// TIA Portal V18 export
VAR_GLOBAL   // PLC tag table "Assigned IO"
   HPU_In AT %I0.0 : "Starter_HPU_IO_In";
   HPU_Out AT %Q0.0 : "Starter_HPU_IO_Out";
   Console_In AT %I200.0 : "Console_IO_In";
   Console_Out AT %Q200.0 : "Console_IO_Out";
   ComFault AT %M20.1 : Bool;
   SystemFault AT %M1.0 : Bool;
   RemConsole_In AT %I500.0 : "RemConsole_IO_In";
   RemConsole_Out AT %Q500.0 : "RemConsole_IO_Out";
   RemConEn AT %M29.6 : Bool;   // Remote console is enable if Aux or TD En and heartbeat is ok
END_VAR
